TYPE ServicesParts :
STRUCT
	///Timing service
	timing: ServicesTiming;
	///The config manager (to load/save/activate configuration data)
	configManager: ConfigManager;
END_STRUCT
END_TYPE

(* stored: Version 1.1.0.1, ProductVersion 3.1.4019.2
   DUT ServicesParts: Id {a900a5d2-8513-44d6-9137-534558976adc} *)
